// TIA Portal V17 export
// export: Created 2024-08-29T18:23:43.2475608Z, ExportSetting WithDefaults, DisplayName Totally Integrated Automation Portal, DisplayVersion V17 Update 7, DisplayName TIA Portal Openness, DisplayVersion V17 Update 7, DisplayName TIA Portal Version Control Interface, DisplayVersion V17, DisplayName SINAMICS Startdrive Advanced, DisplayVersion V17 SP2, DisplayName SINAMICS Startdrive G110M, G120, G120C, G120D, G120P, G115D, DisplayVersion V17 SP2, DisplayName SINAMICS Startdrive G130, G150, S120, S150, SINAMICS MV, S210, DisplayVersion V17 SP2, DisplayName STEP 7 Professional, DisplayVersion V17 Update 7, DisplayName STEP 7 Safety, DisplayVersion V17 Update 6, DisplayName WinCC Advanced / Unified PC, DisplayVersion V17 Update 7
DATA_BLOCK "outputs"   // DB2
{ S7_Optimized_Access := 'TRUE' }
VERSION : 0.1
// stored: AutoNumber false, DBAccessibleFromOPCUA true, DBAccessibleFromWebserver true, IsOnlyStoredInLoadMemory false, IsRetainMemResEnabled false, IsWriteProtectedInAS false, MemoryReserve 0
   VAR RETAIN
      outputSequence : Array[0..32, 0..25] of DInt;   // 32 salidas [modelo, paso]
   END_VAR
   VAR
      activeOutputsReq : Array[0..31] of Bool;
   END_VAR
   VAR RETAIN
      maskSequence : Array[0..32, 0..25] of DInt;   // Máscara de salidas
   END_VAR
   VAR
      activeMask : Array[0..31] of Bool;
      active : DInt := 85;
      outputsActive : Array[0..31] of Bool;
   END_VAR
   VAR RETAIN
      text : Array[0..31] of String;   // Texto HMI de cada salida
   END_VAR
   VAR
      availableNameManipulate : Array[0..8] of String;   // Texto HMI en pagina Manual
      status : Array[0..63] of Bool;
      cylinderDirectionA : Array[0..9] of Bool;   // Variable HMI para activar avance
      cylinderDirectionB : Array[0..9] of Bool;   // Variable HMI para activar retroceso
      cylinderDirectionAActive : Array[0..9] of Bool;   // Variable HMI para enclavamiento avance
      cylinderDirectionBActive : Array[0..9] of Bool;   // Variable HMI para enclavamiento retroceso
      cylinderDirectionAStatus : Array[0..9] of Bool;   // Variable HMI para enclavamiento avance
      cylinderDirectionBStatus : Array[0..9] of Bool;   // Variable HMI para enclavamiento retroceso
      vent : Array[0..9] of Bool;   // Variable HMI para desactivar electroválvula
      cylinderStatus : Array[0..9] of Int;   // Variable HMI para estado de los botones de manipulación
      activateOutput : Array[0..31] of Bool;
      activeAlarm : Bool := FALSE;
      showTextsOutputs : Bool := FALSE;
      cicleTime : Int := 0;
      cicleTimeTimerReset : Bool := FALSE;
      timer1 { S7_SetPoint := 'True'} : TON_TIME;
      timer2 { S7_SetPoint := 'True'} : TON_TIME;
      timer3 { S7_SetPoint := 'True'} : TON_TIME;
      timer4 { S7_SetPoint := 'True'} : TON_TIME;
      timer5 { S7_SetPoint := 'True'} : TON_TIME;
      timer6 { S7_SetPoint := 'True'} : TON_TIME;
      timer7 { S7_SetPoint := 'True'} : TON_TIME;
      timer8 { S7_SetPoint := 'True'} : TON_TIME;
      timer9 { S7_SetPoint := 'True'} : TON_TIME;
      timer10 { S7_SetPoint := 'True'} : TON_TIME;
      timer11 { S7_SetPoint := 'True'} : TON_TIME;
      timer12 { S7_SetPoint := 'True'} : TON_TIME;
      timer13 { S7_SetPoint := 'True'} : TON_TIME;
      timer14 { S7_SetPoint := 'True'} : TON_TIME;
      timer15 { S7_SetPoint := 'True'} : TON_TIME;
      timer16 { S7_SetPoint := 'True'} : TON_TIME;
      timer17 { S7_SetPoint := 'True'} : TON_TIME;
      timer18 { S7_SetPoint := 'True'} : TON_TIME;
      timer19 { S7_SetPoint := 'True'} : TON_TIME;
      timer20 { S7_SetPoint := 'True'} : TON_TIME;
      timer21 { S7_SetPoint := 'True'} : TON_TIME;
      timer22 { S7_SetPoint := 'True'} : TON_TIME;
      timer23 { S7_SetPoint := 'True'} : TON_TIME;
      timer24 { S7_SetPoint := 'True'} : TON_TIME;
      timer25 { S7_SetPoint := 'True'} : TON_TIME;
      timer26 { S7_SetPoint := 'True'} : TON_TIME;
      timer27 { S7_SetPoint := 'True'} : TON_TIME;
      timer28 { S7_SetPoint := 'True'} : TON_TIME;
      timer29 { S7_SetPoint := 'True'} : TON_TIME;
      timer30 { S7_SetPoint := 'True'} : TON_TIME;
      timer31 { S7_SetPoint := 'True'} : TON_TIME;
      "timer" { S7_SetPoint := 'True'} : Array[0..31] of ton_time;
      reset : Bool := FALSE;
      timerReset : Bool := FALSE;
      visibility : Array[0..8] of Bool;
      visualizeCicleTime : Int := 111;
      energysaverTimer { S7_SetPoint := 'True'} : TON_TIME;
      scannerOk : Array[0..5] of Bool;
      scannerLength : Array[0..5] of Int;
      cilinder1 : Bool := TRUE;
      cilinder2 : Bool := TRUE;
      cilinder3 : Bool := TRUE;
      cilinder4 : Bool := FALSE;
      cilinder5 : Bool := FALSE;
      cilinder6 : Bool := FALSE;
      cilinder7 : Bool := FALSE;
      cilinder8 : Bool := FALSE;
   END_VAR
BEGIN
   outputSequence[0,0] := 90;
   outputSequence[0,1] := 85;
   outputSequence[0,2] := 166;
   outputSequence[0,3] := 422;
   outputSequence[0,4] := 681;
   outputSequence[0,5] := 165;
   outputSequence[0,6] := 66726;
   outputSequence[0,7] := 170;
   outputSequence[0,8] := 133289;
   outputSequence[0,9] := 536_871_082;
   outputSequence[0,10] := 90;
   outputSequence[0,11..25] := 0;
   outputSequence[1,0] := 90;
   outputSequence[1,1] := 85;
   outputSequence[1,2] := 166;
   outputSequence[1,3] := 422;
   outputSequence[1,4] := 681;
   outputSequence[1,5] := 165;
   outputSequence[1,6] := 66726;
   outputSequence[1,7] := 170;
   outputSequence[1,8] := 133289;
   outputSequence[1,9] := 536_871_082;
   outputSequence[1,10] := 90;
   outputSequence[1,11..25] := 0;
   outputSequence[2,0] := 90;
   outputSequence[2,1] := 85;
   outputSequence[2,2] := 166;
   outputSequence[2,3] := 422;
   outputSequence[2,4] := 681;
   outputSequence[2,5] := 165;
   outputSequence[2,6] := 66726;
   outputSequence[2,7] := 170;
   outputSequence[2,8] := 133289;
   outputSequence[2,9] := 536_871_082;
   outputSequence[2,10] := 90;
   outputSequence[2,11..25] := 0;
   outputSequence[3,0] := 90;
   outputSequence[3,1] := 85;
   outputSequence[3,2] := 170;
   outputSequence[3,3] := 938;
   outputSequence[3,4] := 170;
   outputSequence[3,5] := 1194;
   outputSequence[3,6..7] := 1193;
   outputSequence[3,8] := 3241;
   outputSequence[3,9] := 80;
   outputSequence[3,10] := 90;
   outputSequence[3,11..25] := 0;
   outputSequence[4,0] := -1_073_741_488;
   outputSequence[4,1] := -956_301_013;
   outputSequence[4,2] := 117_440_810;
   outputSequence[4,3] := -1_073_741_653;
   outputSequence[4,4] := 65715;
   outputSequence[4,5] := 65739;
   outputSequence[4,6] := 171;
   outputSequence[4,7] := 301;
   outputSequence[4,8] := 134_742_317;
   outputSequence[4,9] := 341;
   outputSequence[4,10..25] := 0;
   outputSequence[5,0] := 90;
   outputSequence[5,1] := 89;
   outputSequence[5,2] := 90;
   outputSequence[5,3] := 89;
   outputSequence[5,4..25] := 0;
   outputSequence[6,0] := 90;
   outputSequence[6,1] := 85;
   outputSequence[6,2] := 170;
   outputSequence[6,3] := 938;
   outputSequence[6,4] := 170;
   outputSequence[6,5] := 66730;
   outputSequence[6,6] := 170;
   outputSequence[6,7] := 169;
   outputSequence[6,8] := 133289;
   outputSequence[6,9] := 89;
   outputSequence[6,10..25] := 0;
   outputSequence[7,0] := 90;
   outputSequence[7,1] := 85;
   outputSequence[7,2] := 170;
   outputSequence[7,3] := 938;
   outputSequence[7,4] := 170;
   outputSequence[7,5] := 66726;
   outputSequence[7,6] := 170;
   outputSequence[7,7] := 169;
   outputSequence[7,8] := 133289;
   outputSequence[7,9] := 89;
   outputSequence[7,10..25] := 0;
   outputSequence[8,0] := 90;
   outputSequence[8,1] := 85;
   outputSequence[8,2] := 170;
   outputSequence[8,3] := 938;
   outputSequence[8,4] := 170;
   outputSequence[8,5] := 66726;
   outputSequence[8,6] := 170;
   outputSequence[8,7] := 169;
   outputSequence[8,8] := 133289;
   outputSequence[8,9] := 89;
   outputSequence[8,10..25] := 0;
   outputSequence[9,0] := 336;
   outputSequence[9,1] := 298;
   outputSequence[9,2] := 299;
   outputSequence[9,3] := 171;
   outputSequence[9,4] := 65715;
   outputSequence[9,5] := 65739;
   outputSequence[9,6] := 171;
   outputSequence[9,7] := 301;
   outputSequence[9,8] := 134_742_317;
   outputSequence[9,9] := 341;
   outputSequence[9,10..25] := 0;
   outputSequence[10,0] := 336;
   outputSequence[10,1] := 298;
   outputSequence[10,2] := 299;
   outputSequence[10,3] := 171;
   outputSequence[10,4] := 65715;
   outputSequence[10,5] := 65739;
   outputSequence[10,6] := 171;
   outputSequence[10,7] := 301;
   outputSequence[10,8] := 134_742_317;
   outputSequence[10,9] := 341;
   outputSequence[10,10..25] := 0;
   outputSequence[11,0] := 336;
   outputSequence[11,1] := 298;
   outputSequence[11,2] := 299;
   outputSequence[11,3] := 171;
   outputSequence[11,4] := 65715;
   outputSequence[11,5] := 65739;
   outputSequence[11,6] := 171;
   outputSequence[11,7] := 301;
   outputSequence[11,8] := 134_742_317;
   outputSequence[11,9] := 341;
   outputSequence[11,10..25] := 0;
   outputSequence[12,0] := 336;
   outputSequence[12,1] := 298;
   outputSequence[12,2] := 299;
   outputSequence[12,3] := 171;
   outputSequence[12,4] := 65715;
   outputSequence[12,5] := 65739;
   outputSequence[12,6] := 171;
   outputSequence[12,7] := 301;
   outputSequence[12,8] := 134_742_317;
   outputSequence[12,9] := 341;
   outputSequence[12,10..25] := 0;
   outputSequence[13,0] := 336;
   outputSequence[13,1] := 298;
   outputSequence[13,2] := 299;
   outputSequence[13,3] := 171;
   outputSequence[13,4] := 65715;
   outputSequence[13,5] := 65739;
   outputSequence[13,6] := 171;
   outputSequence[13,7] := 301;
   outputSequence[13,8] := 134_742_317;
   outputSequence[13,9] := 341;
   outputSequence[13,10..25] := 0;
   outputSequence[14,0] := 336;
   outputSequence[14,1] := 117_440_810;
   outputSequence[14,2] := 299;
   outputSequence[14,3] := 171;
   outputSequence[14,4] := 65715;
   outputSequence[14,5] := 65739;
   outputSequence[14,6] := 171;
   outputSequence[14,7] := 301;
   outputSequence[14,8] := 134_742_317;
   outputSequence[14,9] := 341;
   outputSequence[14,10..25] := 0;
   outputSequence[15,0] := 5408;
   outputSequence[15,1..2] := 4768;
   outputSequence[15,3] := 800;
   outputSequence[15,4] := 11040;
   outputSequence[15,5] := 11424;
   outputSequence[15,6] := 4800;
   outputSequence[15,7] := 37568;
   outputSequence[15,8] := 5440;
   outputSequence[15,9..25] := 0;
   outputSequence[16,0] := 336;
   outputSequence[16,1] := 298;
   outputSequence[16,2] := 299;
   outputSequence[16,3] := 171;
   outputSequence[16,4] := 65715;
   outputSequence[16,5] := 65739;
   outputSequence[16,6] := 171;
   outputSequence[16,7] := 301;
   outputSequence[16,8] := 134_742_317;
   outputSequence[16,9] := 341;
   outputSequence[16,10..25] := 0;
   outputSequence[17,0] := 336;
   outputSequence[17,1] := 298;
   outputSequence[17,2] := 299;
   outputSequence[17,3] := 171;
   outputSequence[17,4] := 65715;
   outputSequence[17,5] := 65739;
   outputSequence[17,6] := 171;
   outputSequence[17,7] := 301;
   outputSequence[17,8] := 134_742_317;
   outputSequence[17,9] := 341;
   outputSequence[17,10..25] := 0;
   outputSequence[18,0] := 336;
   outputSequence[18,1] := 117_440_810;
   outputSequence[18,2] := 117_440_811;
   outputSequence[18,3] := 171;
   outputSequence[18,4] := 65715;
   outputSequence[18,5] := 65739;
   outputSequence[18,6] := 171;
   outputSequence[18,7] := 301;
   outputSequence[18,8] := 940_048_685;
   outputSequence[18,9] := 341;
   outputSequence[18,10..25] := 0;
   outputSequence[19,0] := 336;
   outputSequence[19,1] := 298;
   outputSequence[19,2] := 299;
   outputSequence[19,3] := 171;
   outputSequence[19,4] := 65715;
   outputSequence[19,5] := 65739;
   outputSequence[19,6] := 171;
   outputSequence[19,7] := 301;
   outputSequence[19,8] := 134_742_317;
   outputSequence[19,9] := 341;
   outputSequence[19,10..25] := 0;
   outputSequence[20,0..25] := 0;
   outputSequence[21,0..25] := 0;
   outputSequence[22,0..25] := 0;
   outputSequence[23,0..25] := 0;
   outputSequence[24,0..25] := 0;
   outputSequence[25,0..25] := 0;
   outputSequence[26,0..25] := 0;
   outputSequence[27,0..25] := 0;
   outputSequence[28,0..25] := 0;
   outputSequence[29,0..25] := 0;
   outputSequence[30,0..25] := 0;
   outputSequence[31,0..25] := 0;
   outputSequence[32,0..25] := 0;
   activeOutputsReq[0] := FALSE;
   activeOutputsReq[1] := TRUE;
   activeOutputsReq[2] := FALSE;
   activeOutputsReq[3..4] := TRUE;
   activeOutputsReq[5] := FALSE;
   activeOutputsReq[6] := TRUE;
   activeOutputsReq[7..31] := FALSE;
   maskSequence[0,0..25] := 0;
   maskSequence[1,0..25] := 0;
   maskSequence[2,0..25] := 0;
   maskSequence[3,0..4] := 0;
   maskSequence[3,5..8] := 1024;
   maskSequence[3,9..25] := 0;
   maskSequence[4,0] := 6;
   maskSequence[4,1..2] := 8;
   maskSequence[4,3..4] := 117_440_522;
   maskSequence[4,5] := 117_473_282;
   maskSequence[4,6] := 117_440_522;
   maskSequence[4,7] := -134_283_256;
   maskSequence[4,8] := -135_004_161;
   maskSequence[4,9] := 117_440_512;
   maskSequence[4,10..25] := 0;
   maskSequence[5,0] := -11;
   maskSequence[5,1] := -10;
   maskSequence[5,2] := -11;
   maskSequence[5,3] := -10;
   maskSequence[5,4..25] := 0;
   maskSequence[6,0..25] := 0;
   maskSequence[7,0..25] := 0;
   maskSequence[8,0..25] := 0;
   maskSequence[9,0] := 6;
   maskSequence[9,1..4] := 8;
   maskSequence[9,5] := 32768;
   maskSequence[9,6] := 10;
   maskSequence[9,7] := -134_283_256;
   maskSequence[9,8] := -134_742_017;
   maskSequence[9,9..25] := 0;
   maskSequence[10,0] := 6;
   maskSequence[10,1..4] := 8;
   maskSequence[10,5] := 32768;
   maskSequence[10,6] := 10;
   maskSequence[10,7] := -134_283_256;
   maskSequence[10,8] := -134_742_017;
   maskSequence[10,9..25] := 0;
   maskSequence[11,0] := 6;
   maskSequence[11,1..4] := 8;
   maskSequence[11,5] := 32768;
   maskSequence[11,6] := 10;
   maskSequence[11,7] := -134_283_256;
   maskSequence[11,8] := -134_742_017;
   maskSequence[11,9..25] := 0;
   maskSequence[12,0] := 6;
   maskSequence[12,1..4] := 8;
   maskSequence[12,5] := 32768;
   maskSequence[12,6] := 10;
   maskSequence[12,7] := -134_283_256;
   maskSequence[12,8] := -134_742_017;
   maskSequence[12,9..25] := 0;
   maskSequence[13,0] := 6;
   maskSequence[13,1..4] := 8;
   maskSequence[13,5] := 32768;
   maskSequence[13,6] := 10;
   maskSequence[13,7] := -134_283_256;
   maskSequence[13,8] := -134_742_017;
   maskSequence[13,9..25] := 0;
   maskSequence[14,0] := 6;
   maskSequence[14,1..4] := 8;
   maskSequence[14,5] := 32768;
   maskSequence[14,6] := 10;
   maskSequence[14,7] := -134_283_256;
   maskSequence[14,8] := -134_742_017;
   maskSequence[14,9..25] := 0;
   maskSequence[15,0] := 4096;
   maskSequence[15,1..2] := 0;
   maskSequence[15,3] := 32;
   maskSequence[15,4..25] := 0;
   maskSequence[16,0] := 6;
   maskSequence[16,1..4] := 8;
   maskSequence[16,5] := 32768;
   maskSequence[16,6] := 10;
   maskSequence[16,7] := -134_283_256;
   maskSequence[16,8] := -134_742_017;
   maskSequence[16,9..25] := 0;
   maskSequence[17,0] := 6;
   maskSequence[17,1..4] := 8;
   maskSequence[17,5] := 32768;
   maskSequence[17,6] := 10;
   maskSequence[17,7] := -134_283_256;
   maskSequence[17,8] := -134_742_017;
   maskSequence[17,9..25] := 0;
   maskSequence[18,0] := 117_440_518;
   maskSequence[18,1..2] := 8;
   maskSequence[18,3..4] := 117_440_520;
   maskSequence[18,5] := 117_473_280;
   maskSequence[18,6] := 117_440_522;
   maskSequence[18,7] := -134_283_256;
   maskSequence[18,8] := -940_048_385;
   maskSequence[18,9] := 117_440_512;
   maskSequence[18,10..25] := 0;
   maskSequence[19,0] := 6;
   maskSequence[19,1..4] := 8;
   maskSequence[19,5] := 32768;
   maskSequence[19,6] := 10;
   maskSequence[19,7] := -134_283_256;
   maskSequence[19,8] := -134_742_017;
   maskSequence[19,9..25] := 0;
   maskSequence[20,0..25] := 0;
   maskSequence[21,0..25] := 0;
   maskSequence[22,0..25] := 0;
   maskSequence[23,0..25] := 0;
   maskSequence[24,0..25] := 0;
   maskSequence[25,0..25] := 0;
   maskSequence[26,0..25] := 0;
   maskSequence[27,0..25] := 0;
   maskSequence[28,0..25] := 0;
   maskSequence[29,0..25] := 0;
   maskSequence[30,0..25] := 0;
   maskSequence[31,0..25] := 0;
   maskSequence[32,0..25] := 0;
   activeMask[0..31] := FALSE;
   outputsActive[0] := TRUE;
   outputsActive[1] := FALSE;
   outputsActive[2] := TRUE;
   outputsActive[3] := FALSE;
   outputsActive[4] := TRUE;
   outputsActive[5] := FALSE;
   outputsActive[6] := TRUE;
   outputsActive[7..31] := FALSE;
   text[0] := 'CIL BLOQUEO NIDO IZQ EXT';
   text[1] := 'CIL BLOQUEO NIDO IZQ RET';
   text[2] := 'CIL BLOQUEO NIDO DER EXT';
   text[3] := 'CIL BLOQUEO NIDO DER RET';
   text[4] := 'CIL BLOQUEO TRACK DER EXT';
   text[5] := 'CIL BLOQUEO TRACK DER RET';
   text[6] := 'CIL BLOQUEO TRACK IZQ EXT';
   text[7] := 'CIL BLOQUEO TRACK IZQ RET';
   text[8] := 'ESFUERZO IZQ OK CC15010';
   text[9] := 'ESFUERZO DER OK CC15080';
   text[10] := 'DISTANCIA IZQ INSERCION OK SD14160';
   text[11] := 'DISTANCIA DER INSERCION OK SD14120';
   text[12..15] := 'RESERVA';
   text[16] := 'Prueba motor  izq';
   text[17] := 'Prueba motor derecho';
   text[18..28] := 'Reserva';
   text[29] := 'Imprimir';
   text[30..31] := 'Reserva';
   availableNameManipulate[0] := 'Bloqueo nido izq';
   availableNameManipulate[1] := 'Bloqueo nido der';
   availableNameManipulate[2] := 'Bloqueo track der';
   availableNameManipulate[3] := 'Bloqueo track izq';
   availableNameManipulate[4] := 'Spare 4';
   availableNameManipulate[5] := 'Spare 5';
   availableNameManipulate[6..8] := '';
   status[0] := FALSE;
   status[1] := TRUE;
   status[2] := FALSE;
   status[3] := TRUE;
   status[4] := FALSE;
   status[5] := TRUE;
   status[6] := FALSE;
   status[7] := TRUE;
   status[8..28] := FALSE;
   status[29] := TRUE;
   status[30..63] := FALSE;
   cylinderDirectionA[0..9] := FALSE;
   cylinderDirectionB[0..9] := FALSE;
   cylinderDirectionAActive[0..3] := TRUE;
   cylinderDirectionAActive[4..9] := FALSE;
   cylinderDirectionBActive[0..9] := FALSE;
   cylinderDirectionAStatus[0..9] := FALSE;
   cylinderDirectionBStatus[0..9] := FALSE;
   vent[0..9] := FALSE;
   cylinderStatus[0..9] := 0;
   activateOutput[0] := TRUE;
   activateOutput[1] := FALSE;
   activateOutput[2] := TRUE;
   activateOutput[3] := FALSE;
   activateOutput[4] := TRUE;
   activateOutput[5] := FALSE;
   activateOutput[6] := TRUE;
   activateOutput[7..31] := FALSE;
   timer1.PT := T#0MS;
   timer1.IN := FALSE;
   timer2.PT := T#0MS;
   timer2.IN := FALSE;
   timer3.PT := T#0MS;
   timer3.IN := FALSE;
   timer4.PT := T#0MS;
   timer4.IN := FALSE;
   timer5.PT := T#0MS;
   timer5.IN := FALSE;
   timer6.PT := T#0MS;
   timer6.IN := FALSE;
   timer7.PT := T#0MS;
   timer7.IN := FALSE;
   timer8.PT := T#0MS;
   timer8.IN := FALSE;
   timer9.PT := T#0MS;
   timer9.IN := FALSE;
   timer10.PT := T#0MS;
   timer10.IN := FALSE;
   timer11.PT := T#0MS;
   timer11.IN := FALSE;
   timer12.PT := T#0MS;
   timer12.IN := FALSE;
   timer13.PT := T#0MS;
   timer13.IN := FALSE;
   timer14.PT := T#0MS;
   timer14.IN := FALSE;
   timer15.PT := T#0MS;
   timer15.IN := FALSE;
   timer16.PT := T#0MS;
   timer16.IN := FALSE;
   timer17.PT := T#0MS;
   timer17.IN := FALSE;
   timer18.PT := T#0MS;
   timer18.IN := FALSE;
   timer19.PT := T#0MS;
   timer19.IN := FALSE;
   timer20.PT := T#0MS;
   timer20.IN := FALSE;
   timer21.PT := T#0MS;
   timer21.IN := FALSE;
   timer22.PT := T#0MS;
   timer22.IN := FALSE;
   timer23.PT := T#0MS;
   timer23.IN := FALSE;
   timer24.PT := T#0MS;
   timer24.IN := FALSE;
   timer25.PT := T#0MS;
   timer25.IN := FALSE;
   timer26.PT := T#0MS;
   timer26.IN := FALSE;
   timer27.PT := T#0MS;
   timer27.IN := FALSE;
   timer28.PT := T#0MS;
   timer28.IN := FALSE;
   timer29.PT := T#0MS;
   timer29.IN := FALSE;
   timer30.PT := T#0MS;
   timer30.IN := FALSE;
   timer31.PT := T#0MS;
   timer31.IN := FALSE;
   "timer"[0..31].PT := T#0MS;
   "timer"[0..31].IN := FALSE;
   visibility[0] := FALSE;
   visibility[1..3] := TRUE;
   visibility[4..8] := FALSE;
   energysaverTimer.PT := T#16M;
   energysaverTimer.IN := TRUE;
   scannerOk[0..5] := FALSE;
   scannerLength[0] := 0;
   scannerLength[1] := 3;
   scannerLength[2..3] := 7;
   scannerLength[4..5] := 0;
END_DATA_BLOCK
